{attribute addProperty BoxType "EPP6228-0022-0016"}
{attribute addProperty Id "State_Ch1AT %I*USINT811State_Ch2AT %I*USINT812State_Ch3AT %I*USINT813State_Ch4AT %I*USINT814State_Ch5AT %I*USINT815State_Ch6AT %I*USINT816State_Ch7AT %I*USINT817State_Ch8AT %I*USINT818"}
{attribute addProperty CRC "3682114920"}
{attribute addProperty SizeInBites "64"}
{attribute addProperty SizeInBytes "8"}
TYPE DeviceState_Inputs_DB789D68 :
STRUCT
	{attribute addProperty Name "State_Ch1"}
	State_Ch1 AT %I* : USINT;
	{attribute addProperty Name "State_Ch2"}
	State_Ch2 AT %I* : USINT;
	{attribute addProperty Name "State_Ch3"}
	State_Ch3 AT %I* : USINT;
	{attribute addProperty Name "State_Ch4"}
	State_Ch4 AT %I* : USINT;
	{attribute addProperty Name "State_Ch5"}
	State_Ch5 AT %I* : USINT;
	{attribute addProperty Name "State_Ch6"}
	State_Ch6 AT %I* : USINT;
	{attribute addProperty Name "State_Ch7"}
	State_Ch7 AT %I* : USINT;
	{attribute addProperty Name "State_Ch8"}
	State_Ch8 AT %I* : USINT;
END_STRUCT
END_TYPE

(* stored: Version 1.2.0.0, ProductVersion 3.1.4024.9
   DUT DeviceState_Inputs_DB789D68: Id {1be41ce3-ab96-4725-8fa9-2772354fdd80} *)
